// TIA Portal V20 export
FUNCTION_BLOCK "Arms"   // FB430, LAD
{ S7_Optimized_Access := 'TRUE' }
// stored: AutoNumber false, MemoryReserve 100, SetENOAutomatically false
   VAR_INPUT
      InclinometerInput1 : Int;
      Arm1BasePosSens : Bool;
      InclinometerInput2 : Int;
      Arm2BasePosSens : Bool;
      ReqUp : Bool;
      ReqDown : Bool;
      TipSpeed : Int := 15000;
      Kp_Up : Int := 100;
      Kp_Down : Int;
      Ki : Int;
      SetValue : Int := 78;
   END_VAR
   VAR_OUTPUT
      ArmsWorkPos : Bool;
      ArmsClampsOperPos : Bool;
      ArmsBasePos : Bool;
      Arm1 : Int;
      Arm2 : Int;
      Discrepancy : Real;   // absolut discrepancy value between arms
   END_VAR
   VAR
      Arm1AngleValue : Real;
      Arm2AngleValue : Real;
      Arm1BasePos : Bool;
      Arm2BasePos : Bool;
      Arm1WorkPos : Bool;
      Arm2WorkPos : Bool;
      Arm1ClampsOperPos : Bool;
      Arm2ClampsOperPos : Bool;
      Integral : Real;
      MAX_Output : Int := 7468;
      MIN_Output : Int := -7468;
      FilteredDiscrepancy : Real;
      Alpha : Real;
      TipSpeedDown : Int;
      SpeedRampTimerDown { S7_SetPoint := 'True'} : TON_TIME;
      SpeedRampTimerUP { S7_SetPoint := 'True'} : TON_TIME;
      TipSpeedAdjusted { S7_SetPoint := 'True'} : Int;
      SpeedReduction : Int := 3000;
      Delta : Int;
      PrevOutput : Int;
   END_VAR
   VAR_TEMP
      P_term : Int;
      I_term : Int;
      output : LInt;
      "dt" : Real;
      Var1 : Real;
   END_VAR
BEGIN

REGION Network 1: Scale Arm1
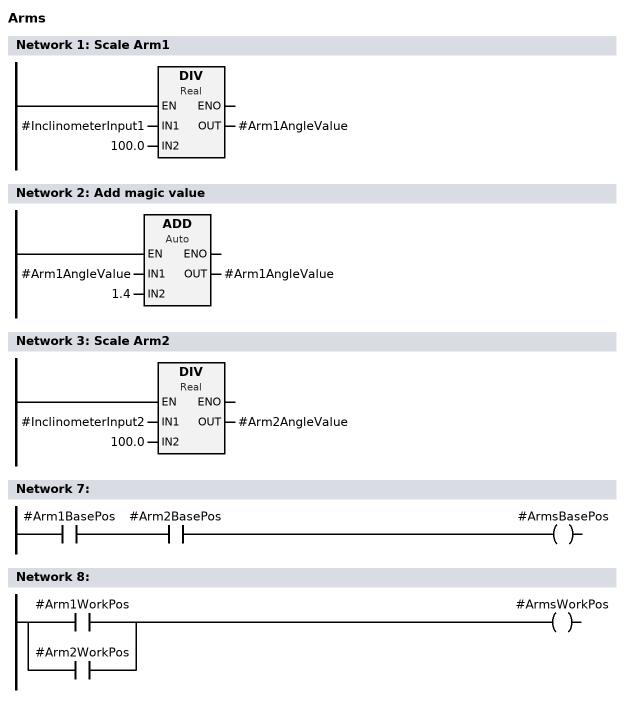
   RUNG wire#powerrail
      { S7_Templates := "SrcType := Real" } Div(in1 := #InclinometerInput1, in2 := 100.0, out => #Arm1AngleValue)
   END_RUNG
   // the same network as SCL:
   #Arm1AngleValue := #InclinometerInput1 / 100.0;
END_REGION

REGION Network 2: Add magic value
   RUNG wire#powerrail
      Add(in1 := #Arm1AngleValue, in2 := 1.4, out => #Arm1AngleValue)
   END_RUNG
   // the same network as SCL:
   #Arm1AngleValue := #Arm1AngleValue + 1.4;
END_REGION

REGION Network 3: Scale Arm2
   RUNG wire#powerrail
      { S7_Templates := "SrcType := Real" } Div(in1 := #InclinometerInput2, in2 := 100.0, out => #Arm2AngleValue)
   END_RUNG
   // the same network as SCL:
   #Arm2AngleValue := #InclinometerInput2 / 100.0;
END_REGION

REGION Network 4 (SCL): Base position Arm1 Arm2
   IF #Arm1AngleValue < 0.05 AND #Arm1BasePosSens THEN
       //BasePos arm 1 
       #Arm1BasePos := TRUE;
   ELSE
       #Arm1BasePos := FALSE;
   END_IF;

   IF #Arm2AngleValue < 0.15 AND #Arm2BasePosSens THEN
       //BasePos arm 2 
       #Arm2BasePos := TRUE;
   ELSE
       #Arm2BasePos := FALSE;
   END_IF;
END_REGION

REGION Network 5 (SCL): Clamps operating position
   #ArmsClampsOperPos := 0;
   IF #Arm1AngleValue > 2 AND #Arm1AngleValue < 3.5 THEN
       //BasePos arm 1 
       #Arm1ClampsOperPos := TRUE;
   ELSE
       #Arm1ClampsOperPos := FALSE;
   END_IF;

   IF #Arm2AngleValue > 2 AND #Arm2AngleValue < 3.5 THEN
       //BasePos arm 2 
       #Arm2ClampsOperPos := TRUE;
   ELSE
       #Arm2ClampsOperPos := FALSE;
   END_IF;

   IF (#Arm1ClampsOperPos OR #Arm2ClampsOperPos) AND ABS(#Discrepancy) < 1.2 THEN
       #ArmsClampsOperPos := 1;
   END_IF;
END_REGION

REGION Network 6 (SCL): Work position Arm1 Arm2
   IF ABS(#Arm1AngleValue - #SetValue) < 1 THEN
       //WorkPos arm 1 
        #Arm1WorkPos := TRUE;
   ELSE
       #Arm1WorkPos := FALSE;
   END_IF;
   IF ABS(#Arm2AngleValue - #SetValue) < 1  THEN
       //WorkPos arm 2 
       #Arm2WorkPos := TRUE;
   ELSE
       #Arm2WorkPos := FALSE;
   END_IF;
END_REGION

REGION Network 7
   RUNG wire#powerrail
      Contact( #Arm1BasePos )
      Contact( #Arm2BasePos )
      Coil( #ArmsBasePos )
   END_RUNG
   // the same network as SCL:
   #ArmsBasePos := #Arm1BasePos AND #Arm2BasePos;
END_REGION

REGION Network 8
   RUNG wire#powerrail
      Contact( #Arm1WorkPos )
      wire#w1
      Coil( #ArmsWorkPos )
   END_RUNG
   RUNG wire#powerrail
      Contact( #Arm2WorkPos )
   END_RUNG wire#w1
   // the same network as SCL:
   #ArmsWorkPos := #Arm1WorkPos OR #Arm2WorkPos;
END_REGION

REGION Network 9 (SCL): discrepancy value between arms
   // -  Arm1 is lower
   // + Arm 1 is higher
   #Discrepancy := #Arm1AngleValue - #Arm2AngleValue;
END_REGION

REGION Network 10 (SCL): MoveArms to workPos by ButtonUp
   // Reset prędkości
   #Arm1 := 0;
   #Arm2 := 0;
   #dt := 0.02; // Czas próbkowania np. 20ms
   #Integral := 0.0;
   #MAX_Output := 3500;
   #MIN_Output := -3500;
   #output := 0;

   // Filtrowanie sygnału z inklinometru (prosty filtr IIR)
   // 

   #SpeedRampTimerUP(IN:= #ReqUp AND "Tippler_DB".Hydraulic_Ready.Q,
                   PT:=T#10s); //4
   IF NOT #SpeedRampTimerUP.Q AND #ReqUp THEN
       #Var1 := INT_TO_REAL(TIME_TO_INT(#SpeedRampTimerUP.ET)) / INT_TO_REAL(TIME_TO_INT(#SpeedRampTimerUP.PT));

       #TipSpeed := 10500 + #Var1 * 9500; //13000 5000
   ELSIF #Arm1AngleValue >= 70.0 THEN
       #TipSpeed := 14500 + 5500 * (81 - #Arm1AngleValue) / 11;
   END_IF;


   #SpeedRampTimerDown(IN := #ReqDown AND "Tippler_DB".Hydraulic_Ready.Q,
                   PT := T#10s); //4
   IF NOT #SpeedRampTimerDown.Q AND #ReqDown THEN
       #Var1 := INT_TO_REAL(TIME_TO_INT(#SpeedRampTimerDown.ET)) / INT_TO_REAL(TIME_TO_INT(#SpeedRampTimerDown.PT));

       #TipSpeed := 10000 + #Var1 * 8000; //10300 7700

   ELSIF #SpeedRampTimerDown.Q AND #ReqDown THEN
       #TipSpeed := 18000;
       IF #Arm1AngleValue <= 7.0 THEN
           #TipSpeed := 10500 + 7500 * (#Arm1AngleValue / 7);
       END_IF;

   END_IF;



   // Jazda w górę
   IF #ReqUp THEN
       #Alpha := 0.05; // tłumienie (0.05 - 0.2 zalecane)
       #FilteredDiscrepancy := #FilteredDiscrepancy + #Alpha * (#Discrepancy - #FilteredDiscrepancy);


       // Arm1: master – jedzie niezależnie do pozycji roboczej
       IF NOT #Arm1WorkPos THEN
           #Arm1 :=#TipSpeed -0;
       END_IF;

       // Arm2: slave – jedzie niezależnie, ale korygowany względem Arm1
       IF NOT #Arm2WorkPos THEN
           // Człon P
           IF NOT "Arm1_UpperClampClosed" THEN
               #Kp_Up := 300;
           END_IF;
           #P_term := REAL_TO_INT(#FilteredDiscrepancy * #Kp_Up);

           // Ograniczenie
           IF #P_term > #MAX_Output THEN
               #output := #MAX_Output;
           ELSIF #P_term < #MIN_Output THEN
               #output := #MIN_Output;
           ELSE
               #output := #P_term;
           END_IF;

           #Delta := #output - #PrevOutput;

           IF #Delta > 10 THEN
               #output := #PrevOutput + 10;
           ELSIF #Delta < -10 THEN
               #output := #PrevOutput - 10;
           END_IF;

           // Zapisz bieżący output jako poprzedni na następny cykl
           #PrevOutput := #output;

           #Arm2 := #Arm1 + #output - 1000;
       END_IF;

       // Jazda w dół
   ELSIF #ReqDown THEN
       #Alpha := 0.02; // tłumienie (0.05 - 0.2 zalecane) //im mniejsze tym bardziej ujednolica
       #FilteredDiscrepancy := #FilteredDiscrepancy + #Alpha * (#Discrepancy - #FilteredDiscrepancy);


       // Arm1: master – jedzie niezależnie do pozycji bazowej
       IF NOT #Arm1BasePos THEN
           IF #Arm1AngleValue > 60 THEN
               #TipSpeedDown := #TipSpeed;
           ELSE
               #TipSpeedDown := #TipSpeed;
           END_IF;
           #Arm1 := - #TipSpeedDown +0;
       END_IF;

       // Arm2: slave – jedzie niezależnie, korygowany względem Arm1
       IF NOT #Arm2BasePos THEN
           #MAX_Output := 3000;
           #MIN_Output := -3000;

           // Człon P
           #P_term := REAL_TO_INT(#FilteredDiscrepancy * #Kp_Down);

           // Ograniczenie
           IF #P_term > #MAX_Output THEN
               #output := #MAX_Output;
           ELSIF #P_term < #MIN_Output THEN
               #output := #MIN_Output;
           ELSE
               #output := #P_term;
           END_IF;

           // Ograniczenie skoku wartości output względem poprzedniego cyklu
           #Delta := #output - #PrevOutput;

           IF #Delta > 4 THEN
               #output := #PrevOutput + 4;
           ELSIF #Delta < -4 THEN
               #output := #PrevOutput - 4;
           END_IF;

           // Zapisz bieżący output jako poprzedni na następny cykl
           #PrevOutput := #output;

           #Arm2 := #Arm1 + #output + 900;
       END_IF;

   END_IF;
END_REGION
END_FUNCTION_BLOCK
